// TwinCAT 3 PLC project tc_mot_example
// ProgramVersion: 3.1.4022.7
// libraries:
//   lcls-twincat-motion, * (SLAC)
//   Tc2_Standard, * (Beckhoff Automation GmbH)
//   Tc2_System, * (Beckhoff Automation GmbH)
//   Tc3_Module, * (Beckhoff Automation GmbH)
// project tree:
//   / PlcTask.TcTTO (not stored)
//   POUs/ Main.TcPOU
// real-time tasks:
//   TASK PlcTask: cycle T#10ms, priority 20, ADS port 350
// motion (NC):
// variable links:
//   tc_mot_example Instance <-> NC-Task 1 SAF/Axes/Example 1 Simulated Working
//     PlcTask Inputs/Main.M1.Axis.NcToPlc <-> Outputs/ToPlc
//     PlcTask Outputs/Main.M1.Axis.PlcToNc <-> Inputs/FromPlc
//   tc_mot_example Instance <-> NC-Task 1 SAF/Axes/Example 2 Simulated Broken
//     PlcTask Inputs/Main.M2.Axis.NcToPlc <-> Outputs/ToPlc
//     PlcTask Outputs/Main.M2.Axis.PlcToNc <-> Inputs/FromPlc
//   tc_mot_example Instance <-> NC-Task 1 SAF/Axes/Example 3 Simulated Limits
//     PlcTask Inputs/Main.M3.Axis.NcToPlc <-> Outputs/ToPlc
//     PlcTask Outputs/Main.M3.Axis.PlcToNc <-> Inputs/FromPlc

// ---- POUs/Main.TcPOU
PROGRAM Main
VAR
    // Simulated motor that is always allowed to move
    {attribute 'pytmc' := '
        pv: PLC:TST:MOT:SIM:01
        field: DESC Simulated Working Motor
    '}
    M1: DUT_MotionStage;
    fbMotion1: FB_MotionStageSim;

    // Simulated motor that is never allowed to move
    {attribute 'pytmc' := '
        pv: PLC:TST:MOT:SIM:02
        field: DESC Simulated Broken Motor
    '}
    M2: DUT_MotionStage;
    fbMotion2: FB_MotionStage;

    // Simulated motor with limits at 0 and 100
    {attribute 'pytmc' := '
        pv: PLC:TST:MOT:SIM:03
        field: DESC Simulated Working Motor With Limits
    '}
    M3: DUT_MotionStage;
    fbMotion3: FB_MotionStage;
    
    // Simulated PPM motor with PMPS
    {attribute 'pytmc' := '
        pv: PLC:TST:MOT:SIM:04
        field: DESC Simulated PPM Motor
    '}
    M4: DUT_MotionStage;
    {attribute 'pytmc' := '
        pv: PLC:TST:MOT:SIM:04
    '}
    fbPPM: FB_PPM;
    
    // PMPS Machinery
    fbArbiterIO: FB_SubSysToArbiter_IO;
    {attribute 'pytmc' := 'pv: PLC:TST:MOT:ARB'}
    fbArbiter: FB_Arbiter(1);
    {attribute 'pytmc' := 'pv: PLC:TST:MOT:FFO:01'}
    fbFFHWO: FB_HardwareFFOutput := (bAutoReset := TRUE);
    
    // Cycle exceed testing
    bCauseExceed: BOOL;
    nDuration: UDINT := 2000000;
    nCounter: UDINT;
    nIndex: UDINT;
    
    fbADSREAD: ADSREAD;
    bRead: BOOL;
    nExceedCount: UDINT;
    
    fbCauseError: FB_CauseNCError;
END_VAR

fbMotion1(stMotionStage := M1);
fbMotion2(stMotionStage := M2);

M3.bHardwareEnable := TRUE;
M3.bPowerSelf := TRUE;
M3.bLimitForwardEnable := M3.Axis.NcToPlc.ActPos < 99.7;
M3.bLimitBackwardEnable := M3.Axis.NcToPlc.ActPos > 0.2;

fbMotion3(stMotionStage := M3);

M4.bHardwareEnable := TRUE;
M4.bPowerSelf := FALSE;
M4.bLimitForwardEnable := TRUE;
M4.bLimitBackwardEnable := TRUE;

fbPPM.nTransitionAssertionID := 16#2FF0;
fbPPM.nUnknownAssertionID := 16#2FF9;
fbPPM.stOut.fPosition := -10;
fbPPM.stOut.bUseRawCounts := FALSE;
fbPPM.stOut.nRequestAssertionID := 16#2FF1;
fbPPM.stOut.stBeamParams := PMPS_GVL.cstFullBeam;
fbPPM.stOut.bValid := TRUE;
fbPPM.stPower.fPosition := -50;
fbPPM.stPower.bUseRawCounts := FALSE;
fbPPM.stPower.nRequestAssertionID := 16#2FF2;
fbPPM.stPower.stBeamParams := PMPS_GVL.cstFullBeam;
fbPPM.stPower.bValid := TRUE;
fbPPM.stYag1.fPosition := -70;
fbPPM.stYag1.bUseRawCounts := FALSE;
fbPPM.stYag1.nRequestAssertionID := 16#2FF3;
fbPPM.stYag1.stBeamParams := PMPS_GVL.cstFullBeam;
fbPPM.stYag1.bValid := TRUE;
fbPPM.stYag2.fPosition := -100;
fbPPM.stYag2.bUseRawCounts := FALSE;
fbPPM.stYag2.nRequestAssertionID := 16#2FF4;
fbPPM.stYag2.stBeamParams := PMPS_GVL.cstFullBeam;
fbPPM.stYag2.bValid := TRUE;

fbPPM(
    stYStage:=M4,
    fbArbiter:=fbArbiter,
    fbFFHWO:=fbFFHWO,
    );
    
fbFFHWO.i_sNetID := '172.21.42.126.1.1';
fbFFHWO.Execute();
fbArbiterIO(
    Arbiter:=fbArbiter,
    fbFFHWO:=fbFFHWO);

IF bCauseExceed THEN
    FOR nIndex := 1 TO nDuration DO
        nCounter := nCounter + 1;
	END_FOR
END_IF

fbADSREAD(
    NETID:='',
    PORT:=350,
    IDXGRP:=16#F200,
    IDXOFFS:=16#100,
    LEN:=SIZEOF(nExceedCount),
    DESTADDR:=ADR(nExceedCount),
    READ:=bRead);
    
fbCauseError(Axis:=M2.Axis);

END_PROGRAM
